(* PLC project CoDeSys External Library Template, WAGO e!COCKPIT e!COCKPIT, author 3S - Smart Software Solutions GmbH *)
(* stored: creationDateTime 2019-10-29T12:37:19.5404406, version 3.5.5.30, modificationDateTime 2019-10-29T12:36:39.3744516, organization 3S - Smart Software Solutions GmbH *)
(* Library project template with all possible element types, docu and a sample project structure *)

TYPE typHarmonogramZdarzenie : STRUCT
  dtCzasRozpoczecia : DT;
  dtCzasZakonczenia : DT;
  sNazwaAtrybutu : STRING(15);
  sWartoscAtrybutu : STRING(15);
END_STRUCT;
END_TYPE
